{attribute 'GeneratedUsingTerminal: EK1122-0000-0018'}
{attribute addProperty BoxType "EK1122-0000-0018"}
{attribute addProperty Id "Beckhoff_EPP4xxxsub_EK1100EK1100_1FC0878B2A_0001_EPP4174_0002_0016EPP4174_D2A7C9B719A_0002_EPP4174_0002_0017EPP4174_D2A7C9B719A_0003_EPP4314_1002_0016EPP4314_1D6CF30B38A_0004_EPP4374_0002_0016EPP4374_6231FEFD36A_0005_EPP4374_0002_0017EPP4374_6231FEFD36A_0006_EPP4374_0002_0018EPP4374_6231FEFD36A_0007_EPP4374_0002_0019EPP4374_6231FEFD36"}
{attribute addProperty CRC "3290525584"}
{attribute addProperty Size "222"}
TYPE Beckhoff_EPP4xxxEK1122_C4216F90 EXTENDS EK1122_1FC0878B :
STRUCT
	{attribute addProperty Name "Beckhoff_EPP4xxxsub_EK1100"}
	Beckhoff_EPP4xxxsub_EK1100 : EK1100_1FC0878B;
	{attribute addProperty Name "A_0001_EPP4174_0002_0016"}
	A_0001_EPP4174_0002_0016 : EPP4174_D2A7C9B7;
	{attribute addProperty Name "A_0002_EPP4174_0002_0017"}
	A_0002_EPP4174_0002_0017 : EPP4174_D2A7C9B7;
	{attribute addProperty Name "A_0003_EPP4314_1002_0016"}
	A_0003_EPP4314_1002_0016 : EPP4314_1D6CF30B;
	{attribute addProperty Name "A_0004_EPP4374_0002_0016"}
	A_0004_EPP4374_0002_0016 : EPP4374_6231FEFD;
	{attribute addProperty Name "A_0005_EPP4374_0002_0017"}
	A_0005_EPP4374_0002_0017 : EPP4374_6231FEFD;
	{attribute addProperty Name "A_0006_EPP4374_0002_0018"}
	A_0006_EPP4374_0002_0018 : EPP4374_6231FEFD;
	{attribute addProperty Name "A_0007_EPP4374_0002_0019"}
	A_0007_EPP4374_0002_0019 : EPP4374_6231FEFD;
END_STRUCT
END_TYPE

(* stored: Version 1.2.0.0, ProductVersion 3.1.4024.9
   DUT Beckhoff_EPP4xxxEK1122_C4216F90: Id {38a05145-beda-48c0-89eb-3e45faa9a98d} *)
